FUNCTION_BLOCK TTestEvent EXTENDS TEventBase 
VAR
    Handler : ITestEventHandler;
END_VAR

METHOD PRIVATE CallHandler
VAR_INPUT
    HandlerBase : IEventHandlerBase;
    EventArgs   : IStreamReader;
END_VAR
IF __QUERYINTERFACE(HandlerBase,Handler) THEN
    Handler.OnCustomEvent(EventArgs);
//ELSE
//    tcl_BaseClasses.F_LogError('Event Handling',F_FormatStringEx1('Error raising %s - invalid handler',EventName));
END_IF
END_METHOD

METHOD IsHandlerSupported : BOOL
VAR_INPUT
    HandlerBase : IEventHandlerBase;
END_VAR
IF __QUERYINTERFACE(HandlerBase,Handler) THEN
    IsHandlerSupported := TRUE;
END_IF
END_METHOD

END_FUNCTION_BLOCK

(* stored: Version 1.1.0.1, ProductVersion 3.1.4024.4
   POU TTestEvent: Id {9bca4868-8dd3-443f-98f1-3cc66debce05}, SpecialFunc None
   Method CallHandler: Id {34fe9b23-b594-43d1-a2d3-e1b9fe18f3fd}
   Method IsHandlerSupported: Id {00bd5167-fde2-46c5-bb8c-119a49f71f25} *)
